(* PLC project bottling_line, Dassault Systèmes ControlBuild 2024x *)
(* stored: creationDateTime 2023-10-03T11:13:41-01:00 *)

PROGRAM panel
  VAR_OUTPUT
    acknowledgePB : BOOL := false;
  END_VAR
  VAR_OUTPUT
    powerUpPB : BOOL := false;
    emergencyStopPB : BOOL := false;
    manual : BOOL := false;
    auto : BOOL := false;
  END_VAR
  VAR_OUTPUT
    startCyclePB : BOOL := false;
    initPB : BOOL := false;
    preparationPB : BOOL := false;
    productionPB : BOOL := false;
    closingPB : BOOL := false;
  END_VAR

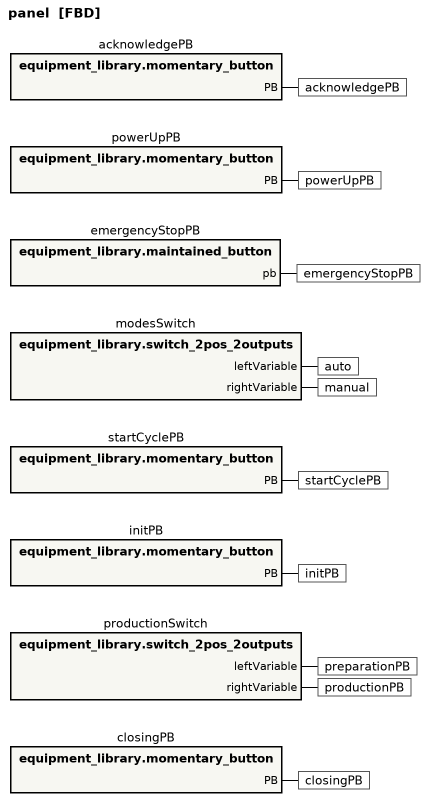
(* FBD diagram, written out as Structured Text *)
acknowledgePB();
acknowledgePB := acknowledgePB.PB;
powerUpPB();
powerUpPB := powerUpPB.PB;
emergencyStopPB();
emergencyStopPB := emergencyStopPB.pb;
modesSwitch();
auto := modesSwitch.leftVariable;
manual := modesSwitch.rightVariable;
startCyclePB();
startCyclePB := startCyclePB.PB;
initPB();
initPB := initPB.PB;
productionSwitch();
preparationPB := productionSwitch.leftVariable;
productionPB := productionSwitch.rightVariable;
closingPB();
closingPB := closingPB.PB;
END_PROGRAM

PROGRAM bottling_line.bottling_line

(* FBD diagram, written out as Structured Text *)
generalPanel();
workingModes(powerUpPB := generalPanel.powerUpPB, emergencyStopPB := generalPanel.emergencyStopPB, manual := generalPanel.manual, auto := generalPanel.auto, acknowledgePB := generalPanel.acknowledgePB);
pumpingTank2(fillingValve := process.valve2, emptyingValve := process.valve4, extractionPump := process.pump2, acknowledgePB := generalPanel.acknowledgePB, autoMode := workingModes.autoMode, manualMode := workingModes.manualMode);
flowsAdd(in1 := pumpingTank1.pumpingFlow, in2 := pumpingTank2.pumpingFlow);
mixing(autoMode := workingModes.autoMode, manualMode := workingModes.manualMode, acknowledgePB := generalPanel.acknowledgePB, fillingValve := process.valve5, hiSpeedAgitator := process.hiSpeedAgitator, loSpeedAgitator := process.loSpeedAgitator, inputFlow := flowsAdd.value);
drive(autoMode := workingModes.autoMode, manualMode := workingModes.manualMode, acknowledgePB := generalPanel.acknowledgePB, load := process.load, evacuate := process.evacuate, convoy := process.convoy, inputFlow := mixing.outputFlow);
process(highLevel1 := pumpingTank1.highLevel, lowLevel1 := pumpingTank1.lowLevel, highLevel2 := pumpingTank2.highLevel, lowLevel2 := pumpingTank2.lowLevel, highLevel3 := mixing.highLevel, lowLevel3 := mixing.lowLevel, startCyclePB := generalPanel.startCyclePB, initPB := generalPanel.initPB, preparationPB := generalPanel.preparationPB, productionPB := generalPanel.productionPB, closingPB := generalPanel.closingPB, pulseGenerator := drive.pulse, bottleFilled := drive.bottleFilled, bottlePresent := drive.bottlePresent);
pumpingTank1(fillingValve := process.valve1, emptyingValve := process.valve3, extractionPump := process.pump1, acknowledgePB := generalPanel.acknowledgePB, autoMode := workingModes.autoMode, manualMode := workingModes.manualMode);
END_PROGRAM
